{attribute 'qualified_only'}
{attribute 'strict'}
TYPE InsertionDirection :
(
	IN,
	OUT,
	
	size
);
END_TYPE

(* stored: Version 1.1.0.1, ProductVersion 3.1.4024.11
   DUT InsertionDirection: Id {7f336cec-9c26-404f-a199-b42cb756868d} *)
